(*
SPDX-FileCopyrightText: © 2026 Oleksandr Tiutyk <trofimich@gmail.com>
SPDX-License-Identifier: MIT
License: https://opensource.org/license/mit
*)

FUNCTION_BLOCK TrySetLightActionDescriptor EXTENDS TOF_Core.Object IMPLEMENTS ITrySetLightActionDescriptor
VAR_STAT
	//! <summary>Class name shared by all instances of this function block.</summary>
	{attribute 'hide'} 
	_ClassName : STRING := __POUNAME();
END_VAR
VAR
	{attribute 'hide'} 
	_Name : WSTRING := "TrySetLight";

	{attribute 'hide'} 
	_NewColor : TRAFFIC_LIGHT_COLOR;
END_VAR

{attribute 'monitoring' := 'call'}
PROPERTY ClassName : REFERENCE TO STRING
GET
ClassName REF= _ClassName;
END_GET
END_PROPERTY

{attribute 'monitoring' := 'call'}
PROPERTY FINAL Name : REFERENCE TO WSTRING
GET
Name REF= _Name;
END_GET
END_PROPERTY

{attribute 'monitoring' := 'call'}
PROPERTY NamespaceName : REFERENCE TO STRING
GET
NamespaceName REF= CurrentNamespace.Name;
END_GET
END_PROPERTY

{attribute 'monitoring' := 'call'}
PROPERTY FINAL NewColor : TRAFFIC_LIGHT_COLOR
GET
NewColor := _NewColor;
END_GET
SET
_NewColor := NewColor;
END_SET
END_PROPERTY

{attribute 'monitoring' := 'call'}
PROPERTY SelfSize : ULINT
GET
SelfSize := XSIZEOF(THIS^);
END_GET
END_PROPERTY

END_FUNCTION_BLOCK

(* stored: Version 1.1.0.1
   POU TrySetLightActionDescriptor: Id {e5614d06-bf7e-4e05-8f0a-e1a0fdcc6367}, SpecialFunc None
   Property ClassName: Id {589e6d42-30cd-445a-9ce8-1ce8d373cc55}
   Get Get: Id {3745626b-3081-4ac7-b507-543269643fc7}
   Property Name: Id {b92f3ebb-0983-4208-952a-94a86711c569}
   Get Get: Id {db4d9deb-be91-467a-a501-96d118b4e1bb}
   Property NamespaceName: Id {8bf1c522-4450-44a6-8cf0-5fbfa342cdd1}
   Get Get: Id {90a1151b-b88c-42bc-be24-0b319da48a6d}
   Property NewColor: Id {00fa84a3-d42b-4b54-a917-f57b41aa82a9}
   Get Get: Id {0d3b551e-694f-4be1-9622-32b2592e0424}
   Set Set: Id {870f3143-347e-4964-938a-8cf1d87644a3}
   Property SelfSize: Id {82ef8ec6-f6f6-477f-8220-8357c3045bb0}
   Get Get: Id {13e8fa12-ea1d-4534-abfe-06387a659075} *)
